(* CODESYS project reflex2.project

Project tree, tasks and I/O mapping:
  Device : CODESYS Control Win V3, 3S - Smart Software Solutions GmbH, order no. 305021, version 3.5.8.10
    application Application
      libraries: Standard, * (System); BASIC, 3.31 (OSCAT)
      task MainTask (cyclic, interval t#20ms, priority 1) calls PLC_PRG
      program PLC_PRG [ST]
      visualisation Visualization
  libraries: VisuSymbols, 3.5.8.0 (System)
  text list GlobalTextList
*)

// Device/Application/PLC_PRG
PROGRAM PLC_PRG
VAR
	set: INT;
	set2: INT;
	last: INT;
	low: INT;
	high: INT;
	
	tim: INT;
	tim2: INT;
	
	x: ARRAY [1..10] OF BOOL;
	t1: ARRAY [1..15] OF TON;
	t2: TOF;
	t3: TON;
	t4: TON;
	
	control: ARRAY [1..4] OF BOOL;
	switch: ARRAY [1..4] OF BOOL;
	
	points: INT;
	
	start: BOOL;
	xx: INT;
	y: INT;
END_VAR

xx := RDM2(last:=0,low:=1,high:=2);
IF((xx = 1)OR(xx = 2)) THEN
	start := TRUE;
END_IF

t1[1](IN:=start,PT:=T#1MS);
x[1] := t1[1].Q;

IF(x[1] = FALSE) THEN
	low := 1;
	high := 4;
	control[1] := FALSE;
	control[2] := FALSE;
	control[3] := FALSE;
	control[4] := FALSE;
	start := FALSE;
	tim2 := 0;
END_IF
IF(x[1] = TRUE) THEN
	low := set;
	high := set;
	x[2] := TRUE;
	x[3] := FALSE;
	start := FALSE;
	tim2 := 0;
END_IF
set := RDM2(last:=0,low:=low,high:=high);

IF(x[2] = TRUE) THEN
	control[set] := TRUE;
END_IF

t3(IN:=control[set],PT:=T#1MS);
x[3] := t3.Q;

IF(x[3] = TRUE) THEN
	x[2] := FALSE;
	x[4] := FALSE;
END_IF

t2(IN:=x[2],PT:=T#5000MS);		// 1300ms
control[set] := t2.Q;
tim := TIME_TO_INT(t2.ET);

IF(tim = 5000) THEN
	x[4] := TRUE;
END_IF

t4(IN:=x[4], PT:=T#10S);
X[5] := T4.Q;
tim2 := TIME_TO_INT(t4.ET);

IF((tim2 < 10000) AND (switch[set] = TRUE)) THEN
	switch[set] := FALSE;
	points := points + 1;
END_IF

IF(tim2 = 10000) THEN
	start := TRUE;
	tim := 0;
	x[1] := FALSE;
END_IF

END_PROGRAM

// Device/Application/Visualization
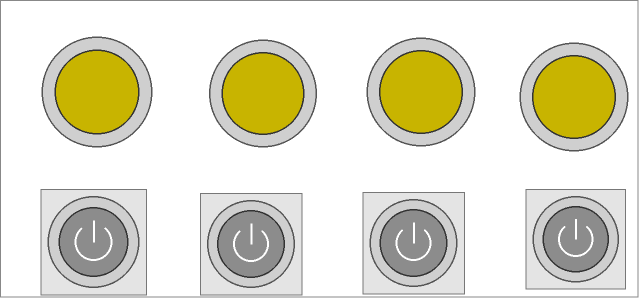
VISUALIZATION Visualization  // 639x298
    Lamp1 (27,28 140x128), variable: PLC_PRG.control[1], style: Lamp-Lamp1-Yellow
    Lamp1 (193,31 140x125), variable: PLC_PRG.control[2], style: Lamp-Lamp1-Yellow
    Lamp1 (352,29 138x126), variable: PLC_PRG.control[3], style: Lamp-Lamp1-Yellow
    Lamp1 (511,32 126x130), variable: PLC_PRG.control[4], style: Lamp-Lamp1-Yellow
    PowerSwitch (36,189 115x106), variable: PLC_PRG.switch[1], behaviour: TOGGLE, style: Switch-PowerSwitch-Gray
    PowerSwitch (200,192 102x104), variable: PLC_PRG.switch[2], behaviour: TOGGLE, style: Switch-PowerSwitch-Gray
    PowerSwitch (362,192 103x102), variable: PLC_PRG.switch[3], behaviour: TOGGLE, style: Switch-PowerSwitch-Gray
    PowerSwitch (523,189 105x100), variable: PLC_PRG.switch[4], behaviour: TOGGLE, style: Switch-PowerSwitch-Gray
END_VISUALIZATION
